INTERFACE ITF_Component2_HMI_Connector_Command EXTENDS ITF_BaseComponent_HMI_Connector_Command

END_INTERFACE

(* stored: Version 1.1.0.1
   Itf ITF_Component2_HMI_Connector_Command: Id {1c28deed-9c36-07dc-338a-081032add8f0} *)
